Fanuc TP program (LS listing): UP101.LS

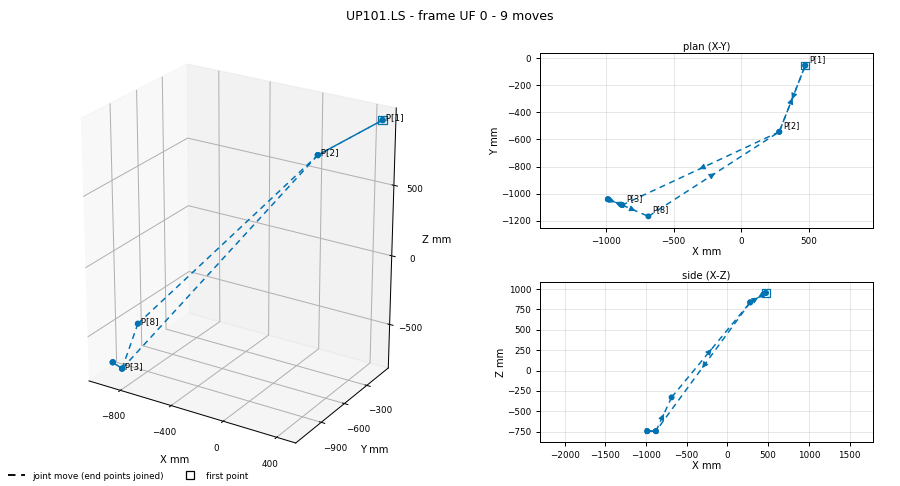
[picture p0: tool path of UP101.LS in frame UF 0, 9 of 10 moves have a stored position in this frame; points joined in program order, loops and branches not executed]
/PROG  UP101
/ATTR
OWNER		= AUROM;
COMMENT		= "Fresado";
PROG_SIZE	= 4718;
CREATE		= DATE 96-03-15  TIME 09:24:00;
MODIFIED	= DATE 23-11-27  TIME 16:22:20;
FILE_NAME	= UP101;
VERSION		= 0;
LINE_COUNT	= 17;
MEMORY_SIZE	= 8602;
PROTECT		= READ_WRITE;
TCD:  STACK_SIZE	= 500,
      TASK_PRIORITY	= 50,
      TIME_SLICE	= 0,
      BUSY_LAMP_OFF	= 0,
      ABORT_REQUEST	= 0,
      PAUSE_REQUEST	= 0;
DEFAULT_GROUP	= 1,1,1,1,*;
CONTROL_CODE	= 00000000 00000000;
/APPL
/MN
   1:  UTOOL_NUM=1 ;
   2:  UFRAME_NUM=0 ;
   3:  PAYLOAD[1] ;
   4:J P[1] 100% CNT0 ACC100 TB    .10sec,P-SPS    ;
      1:  TC_ONLINE (ON) ;
      2:  DO[23]=OFF ;
      3:  CALL MAKRO050    ;
      4:  !Lib. de Herramientas ;
      5:  DO[80]=ON ;
      6:  DO[79]=ON ;
      7:  !Lib. de Anticolisiones ;
      8:  DO[41]=ON ;
      9:  DO[42]=ON ;
     10:  DO[43]=ON ;
     11:  DO[44]=ON ;
     12:  !Apagar Pos. Base ;
     13:  DO[15]=OFF ;
     14:  !Robot en Trayectoria ;
     15:  DO[16]=ON ;
     16:  !Ap. Med. Ant/Dsp. Fresar ;
     17:  DO[756]=OFF ;
     18:  DO[757]=OFF ;
     19:  CALL VW_USER(Basic1,EZSP,Nr1 Service,ProgNr=31, , ,S-Punkt=31, ,EIN/AUS=1) ;
     20:  WAIT    .10(sec) ;
     21:  !Fresado Normal ;
     22:  F[79]=((DI[786] AND !DI[788]) OR F[298] OR (!DI[786] AND !DI[788] AND DO[11]) OR (!DI[788] AND DI[130])) ;
     23:  !Fresado Inicial ;
     24:  F[78]=(DI[788] AND !F[79]) ;
     25:  WAIT (DI[23])    ;
     26:  DO[23]=ON ;
     27:  TC_ONLINE (M[30] AND M[95]) ;
       ------ ;
   5:J P[2] 100% CNT100 ACC100 TB   0.00sec,P-SPS    ;
      1:  TC_ONLINE (M[30] AND M[95]) ;
       ------ ;
   6:J P[3] 100% CNT100 ACC100 TB   0.00sec,P-SPS    ;
      1:  TC_ONLINE (M[30] AND M[95]) ;
       ------ ;
   7:J P[4] 100% CNT0 ACC100 TB    .10sec,P-SPS    ;
      1:  TC_ONLINE (ON) ;
      2:  DO[23]=OFF ;
      3:  WAIT (DI[23])    ;
      4:  DO[23]=ON ;
      5:  TC_ONLINE (M[30] AND M[95]) ;
       ------ ;
   8:  !Posicion de Fresado ;
   9:J P[5] 100% CNT0 ACC100 TB    .10sec,P-SPS Tool_Offset,PR[11] Offset,PR[12]    ;
      1:  TC_ONLINE (ON) ;
      2:  DO[23]=OFF ;
      3:  CALL VW_USER(Basic1,EZSP,Nr1 Service,ProgNr=31, , ,S-Punkt=31, ,EIN/AUS=1) ;
      4:  !Sel. de Pistola ;
      5:  F[64]=(ON) ;
      6:  F[65]=(OFF) ;
      7:  F[66]=(OFF) ;
      8:  F[67]=(OFF) ;
      9:  DO[130]=ON ;
     10:  GO[2]=(R[197]+23) ;
     11:  IF (F[78] OR F[79]),CALL MAKRO082 ;
     12:  DO[130]=OFF ;
     13:  WAIT (DI[23])    ;
     14:  DO[23]=ON ;
     15:  TC_ONLINE (M[30] AND M[95]) ;
       ------ ;
  10:J P[6] 100% CNT0 ACC100 TB    .10sec,P-SPS    ;
      1:  TC_ONLINE (ON) ;
      2:  DO[23]=OFF ;
      3:  WAIT (DI[23])    ;
      4:  DO[23]=ON ;
      5:  TC_ONLINE (M[30] AND M[95]) ;
       ------ ;
  11:J P[7] 100% CNT100 ACC100 TB   0.00sec,P-SPS    ;
      1:  TC_ONLINE (M[30] AND M[95]) ;
       ------ ;
  12:J P[8] 100% CNT100 ACC100 TB   0.00sec,P-SPS    ;
      1:  TC_ONLINE (M[30] AND M[95]) ;
       ------ ;
  13:  !Inic. Med ;
  14:J P[9] 100% CNT100 ACC100 TB   0.00sec,P-SPS    ;
      1:  TC_ONLINE (ON) ;
      2:  DO[715]=ON ;
      3:  DO[757]=ON ;
      4:  TC_ONLINE (M[30] AND M[95]) ;
       ------ ;
  15:  !Fin de Med. ;
  16:  !Posicion Base ;
  17:J P[10] 100% CNT0 ACC100 TB    .10sec,P-SPS    ;
      1:  TC_ONLINE (ON) ;
      2:  DO[23]=OFF ;
      3:  CALL MAKRO083    ;
      4:  IF (F[78] AND !F[79] AND F[335]),CALL MAKRO087 ;
      5:  CALL VW_USER(Basic1,EZSP,Nr1 Service,ProgNr=41, , ,S-Punkt=41, ,EIN/AUS=F[78]) ;
      6:  CALL VW_USER(Basic1,EZSP,Nr1 Service,ProgNr=51, , ,S-Punkt=51, ,EIN/AUS=F[79]) ;
      7:  IF (!F[85] AND !F[86]),CALL MAKRO080 ;
      8:  WAIT (!F[298] OR (DI[777] AND F[298]) OR DI[26] OR (F[298] AND F[749]))    ;
      9:  WAIT (DI[23])    ;
     10:  DO[23]=ON ;
     11:  TC_ONLINE (M[30] AND M[95]) ;
       ------ ;
/POS
P[1]{
   GP1:
	UF : 0, UT : 1,		CONFIG : 'N U T, 0, 0, 0',
	X =   471.294  mm,	Y =   -54.798  mm,	Z =   952.831  mm,
	W =  -172.162 deg,	P =   -29.440 deg,	R =   -25.722 deg
   GP2:
	UF : 0, UT : 1,
	J1=   100.000  mm
   GP3:
	UF : 0, UT : 1,
	J1=     0.000  mm
   GP4:
	UF : 0, UT : 1,
	J1=     0.000  mm
};
P[2]{
   GP1:
	UF : 0, UT : 1,		CONFIG : 'N U T, 0, 0, 0',
	X =   279.805  mm,	Y =  -543.711  mm,	Z =   837.250  mm,
	W =  -171.122 deg,	P =   -33.846 deg,	R =   -81.011 deg
   GP2:
	UF : 0, UT : 1,
	J1=   100.000  mm
   GP3:
	UF : 0, UT : 1,
	J1=     0.000  mm
   GP4:
	UF : 0, UT : 1,
	J1=     0.000  mm
};
P[3]{
   GP1:
	UF : 0, UT : 1,		CONFIG : 'N U T, 0, 0, 0',
	X =  -878.846  mm,	Y = -1084.236  mm,	Z =  -744.811  mm,
	W =   103.402 deg,	P =   -89.253 deg,	R =  -125.257 deg
   GP2:
	UF : 0, UT : 1,
	J1=   100.000  mm
   GP3:
	UF : 0, UT : 1,
	J1=     0.000  mm
   GP4:
	UF : 0, UT : 1,
	J1=     0.000  mm
};
P[4]{
   GP1:
	UF : 0, UT : 1,		CONFIG : 'N U T, 0, 0, 0',
	X =  -983.518  mm,	Y = -1040.266  mm,	Z =  -744.430  mm,
	W =   103.408 deg,	P =   -89.253 deg,	R =  -125.212 deg
   GP2:
	UF : 0, UT : 1,
	J1=   101.400  mm
   GP3:
	UF : 0, UT : 1,
	J1=     0.000  mm
   GP4:
	UF : 0, UT : 1,
	J1=     0.000  mm
};
P[5]{
   GP1:
	UF : 0, UT : 1,		CONFIG : 'N U T, 0, 0, 0',
	X =  -986.917  mm,	Y = -1042.024  mm,	Z =  -708.503  mm,
	W =   157.856 deg,	P =   -89.132 deg,	R =  -179.729 deg
   GP2:
	UF : 0, UT : 1,
	J1=    21.300  mm
   GP3:
	UF : 0, UT : 1,
	J1=     0.000  mm
   GP4:
	UF : 0, UT : 1,
	J1=     0.000  mm
};
P[6]{
   GP1:
	UF : 0, UT : 1,		CONFIG : 'N U T, 0, 0, 0',
	X =  -985.281  mm,	Y = -1041.542  mm,	Z =  -745.158  mm,
	W =   103.385 deg,	P =   -89.253 deg,	R =  -125.241 deg
   GP2:
	UF : 0, UT : 1,
	J1=   100.000  mm
   GP3:
	UF : 0, UT : 1,
	J1=     0.000  mm
   GP4:
	UF : 0, UT : 1,
	J1=     0.000  mm
};
P[7]{
   GP1:
	UF : 0, UT : 1,		CONFIG : 'N U T, 0, 0, 0',
	X =  -878.846  mm,	Y = -1084.236  mm,	Z =  -744.811  mm,
	W =   103.402 deg,	P =   -89.253 deg,	R =  -125.257 deg
   GP2:
	UF : 0, UT : 1,
	J1=   100.000  mm
   GP3:
	UF : 0, UT : 1,
	J1=     0.000  mm
   GP4:
	UF : 0, UT : 1,
	J1=     0.000  mm
};
P[8]{
   GP1:
	UF : 0, UT : 1,		CONFIG : 'N U T, 0, 0, 0',
	X =  -685.598  mm,	Y = -1167.421  mm,	Z =  -329.487  mm,
	W =   103.374 deg,	P =   -89.253 deg,	R =  -125.230 deg
   GP2:
	UF : 0, UT : 1,
	J1=   100.000  mm
   GP3:
	UF : 0, UT : 1,
	J1=     0.000  mm
   GP4:
	UF : 0, UT : 1,
	J1=     0.000  mm
};
P[9]{
   GP1:
	UF : 0, UT : 1,		CONFIG : 'N U T, 0, 0, 0',
	X =   279.805  mm,	Y =  -543.712  mm,	Z =   837.249  mm,
	W =  -171.122 deg,	P =   -33.846 deg,	R =   -81.011 deg
   GP2:
	UF : 0, UT : 1,
	J1=   100.000  mm
   GP3:
	UF : 0, UT : 1,
	J1=     0.000  mm
   GP4:
	UF : 0, UT : 1,
	J1=     0.000  mm
};
P[10]{
   GP1:
	UF : 0, UT : 1,		CONFIG : 'N U T, 0, 0, 0',
	X =   471.294  mm,	Y =   -54.798  mm,	Z =   952.831  mm,
	W =  -172.162 deg,	P =   -29.440 deg,	R =   -25.722 deg
   GP2:
	UF : 0, UT : 1,
	J1=   100.000  mm
   GP3:
	UF : 0, UT : 1,
	J1=     0.000  mm
   GP4:
	UF : 0, UT : 1,
	J1=     0.000  mm
};
/END
